{attribute 'qualified_only'}
VAR_GLOBAL
	bEStopOK			: BOOL;
END_VAR

(* stored: Version 1.1.0.1, ProductVersion 3.1.4024.11
   GVL Safety: Id {15e21265-a001-476a-aefc-148bcfd69842} *)
